// TIA Portal V18 export
VAR_GLOBAL   // PLC tag table "Default tag table"
   pbStart AT %M10.0 : Bool;
   pbSTop AT %M10.1 : Bool;
   Lamp AT %M20.0 : Bool;
   NewTagTest AT %M20.1 : Bool;
END_VAR
